{attribute 'qualified_only'}
TYPE ENU_DT0800EN02 :
(
	Default_watchdog_value := 0,
	Watchdog_ramp,
	Last_output_value
);
END_TYPE

(* stored: Version 1.1.0.1, ProductVersion 3.1.4024.6
   DUT ENU_DT0800EN02: Id {e931dc27-7946-0f58-3d0d-08197093bd2c} *)
